// TwinCAT 3 PLC project Binaire_weergave
// ProgramVersion: 3.1.4024.0
// libraries:
//   Tc2_Standard, * (Beckhoff Automation GmbH)
//   Tc2_System, * (Beckhoff Automation GmbH)
//   Tc3_Module, * (Beckhoff Automation GmbH)
// project tree:
//   / PlcTask.TcTTO
//   POUs/ MAIN.TcPOU
// (motion and I/O tree: see PLC project potentiometer_inlezen)
// real-time tasks:
//   TASK PlcTask: cycle T#10ms, priority 20, ADS port 350
//   TASK PlcTask1: cycle T#10ms, priority 21, ADS port 351
//   TASK PlcTask2: cycle T#10ms, priority 22, ADS port 352
//   TASK PlcTask3: cycle T#10ms, priority 26, ADS port 353
//   TASK PlcTask4: cycle T#10ms, priority 25, ADS port 354
//   TASK PlcTask5: cycle T#10ms, priority 24, ADS port 355
//   TASK PlcTask6: cycle T#10ms, priority 23, ADS port 356
//   TASK PlcTask7: cycle T#10ms, priority 27, ADS port 357

CONFIGURATION Binaire_weergave
    RESOURCE PLC ON TwinCAT3
        TASK PlcTask(INTERVAL := T#10ms, PRIORITY := 25);
        PROGRAM MAIN WITH PlcTask : MAIN;
    END_RESOURCE
END_CONFIGURATION

// ---- POUs/MAIN.TcPOU
PROGRAM MAIN
VAR
	
    fPotmeter: INT := 0; // Gemeten waarde van potentiometer (0 tot 32767)
    bValue: BYTE; // Geconverteerde waarde (0 tot 15)

END_VAR

bValue := TO_BYTE((fPotmeter * 15) / 32767);

END_PROGRAM
